Yaskawa INFORM job: HOME_A.JBI

/JOB
//NAME HOME_A
///FOLDERNAME MASTER
//POS
///NPOS 0,0,0,0,0,1
///TOOL 0
///POSTYPE PULSE
///PULSE
EX00040=-389729
//INST
///DATE 2021/10/29 11:48
///ATTR SC,RO
///GROUP1 ST1
NOP
'*******************************
'THIS JOB HOMES POSITIONER SIDE
'A TO THE ROBOT, SIDE B TO LOAD
'WITHOUT AFFECTING THE TOOLING.
'********************************
MOVJ EX040 VJ=5.00
END
